FUNCTION_BLOCK SS3_ifb_ps_flipper (* Composite FB wrapping other FBs *)
  (* Standard: 61499-2 *)
  (* Version 1.0, 2025-05-26, PS_Transformer_for_Unknown *)
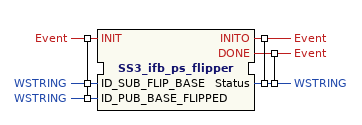
  EVENT_INPUT
    INIT WITH ID_SUB_FLIP_BASE, ID_PUB_BASE_FLIPPED; (* Initialization Request *)
  END_EVENT
  EVENT_OUTPUT
    INITO WITH Status; (* Initialization Confirm *)
    DONE WITH Status; (* Execution Confirmation *)
  END_EVENT
  VAR_INPUT
    ID_SUB_FLIP_BASE : WSTRING;
    ID_PUB_BASE_FLIPPED : WSTRING;
  END_VAR
  VAR_OUTPUT
    Status : WSTRING; (* Output event qualifier *)
  END_VAR
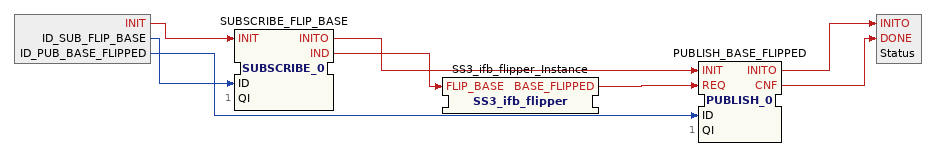
  FBS
    SS3_ifb_flipper_Instance : SS3_ifb_flipper;
    SUBSCRIBE_FLIP_BASE : SUBSCRIBE_0(QI := 1);
    PUBLISH_BASE_FLIPPED : PUBLISH_0(QI := 1);
  END_FBS
  EVENT_CONNECTIONS
    INIT TO SUBSCRIBE_FLIP_BASE.INIT;
    SUBSCRIBE_FLIP_BASE.INITO TO PUBLISH_BASE_FLIPPED.INIT;
    PUBLISH_BASE_FLIPPED.INITO TO INITO;
    SUBSCRIBE_FLIP_BASE.IND TO SS3_ifb_flipper_Instance.FLIP_BASE;
    SS3_ifb_flipper_Instance.BASE_FLIPPED TO PUBLISH_BASE_FLIPPED.REQ;
    PUBLISH_BASE_FLIPPED.CNF TO DONE;
  END_CONNECTIONS
  DATA_CONNECTIONS
    ID_SUB_FLIP_BASE TO SUBSCRIBE_FLIP_BASE.ID;
    ID_PUB_BASE_FLIPPED TO PUBLISH_BASE_FLIPPED.ID;
  END_CONNECTIONS
END_FUNCTION_BLOCK
